PowerOn=0
Idle=1
上下出=2
檢查開始=3
上下回=4
*************************************************************************)
(*************************************************************************
異常碼
急停=1
氣缸=2
檢查NG=3
*************************************************************************)
//*************************************************************************
//本站狀態判斷
IF IndexData[2].OKFlag[2]
	OR IndexData[2].NGFlag[2] THEN
	IndexData[2].FinishFlag[2]:=TRUE;
END_IF;
//前站狀態判斷
IF  	IndexData[2].NGFlag[1] THEN
	IndexData[2].NGFlag[1]:=TRUE;
END_IF;
//本站關閉判斷
IF DisablePB[2] AND IndexData[2].FinishFlag[1] AND IndexData[2].OKFlag[1] AND NOT(IndexData[2].NGFlag[1]) THEN
	IndexData[2].OKFlag[2]:=TRUE;
END_IF;

Rtrig_test(CLK:=TestPB[2]);
//PowerOn=0
IF NOT(SystemReadyStatus AND AutoStatus AND NOT(ErrorStatus[2]) AND NOT(Error_PB_EStop)) THEN
	Autoflow:=0;
END_IF;
	//EStop異常碼
	(*IF Error_PB_Estop AND NOT(IndexData[4].FinishFlag[4]) AND IndexData[4].OkFlag[1] THEN
		IndexData[4].NGFlag[4]:=TRUE;
		IndexData[4].ErrorLog[4]:=1;
	END_IF;*)
	//Error異常碼
	(*IF ErrorStatus[4] AND NOT(IndexData[4].FinishFlag[4]) AND IndexData[4].OkFlag[1] THEN
		IndexData[4].NGFlag[4]:=TRUE;
		IndexData[4].ErrorLog[4]:=2;
	END_IF;*)
//Idle=1
IF AutoFlow=0 AND SystemReadyStatus AND AutoStatus AND NOT(ErrorStatus[2]) AND NOT(Error_PB_EStop) THEN
	AutoFlow:=1;
END_IF;

IF Autoflow=4 AND LS_S2_UpDownBack THEN
	Autoflow:=1;
END_IF;

//上下出=2
IF Autoflow=1
	AND AutoStatus
	AND NOT(DisablePB[2])
	AND LS_S2_UpDownBack
	AND (MachineRunStatus AND NOT(IndexData[2].FinishFlag[2]) AND IndexData[2].FinishFlag[1] AND IndexData[2].OKFlag[1] AND NOT(IndexData[2].NGFlag[1])
	OR Rtrig_test.Q) THEN
	Autoflow:=2;
END_IF;

//檢查開始=3
IF Autoflow=2 AND NOT(LS_S2_UpDownBack) THEN
	Autoflow:=3;
END_IF;
TON1(In:=Autoflow=3 AND LS_S2_UpDownOut, PT:=t#500ms);		//OK
TON2(In:=Autoflow=3 AND NOT(LS_S2_UpDownOut), PT:=t#2000ms);		//NG
//上下回=4
IF Autoflow=3 AND TON1.Q THEN
	IndexData[2].OKFlag[2]:=TRUE;
	IndexData[2].NGFlag[2]:=FALSE;
	Autoflow:=4;
END_IF;

IF Autoflow=3 AND TON2.Q THEN
	IndexData[2].OKFlag[2]:=FALSE;
	IndexData[2].NGFlag[2]:=TRUE;
	IndexData[2].ErrorLog[2]:=3;
	Autoflow:=4;
END_IF;

//*************************************************************************
//手動
//上下電磁閥
R_TRIG_1[0](CLK:=HMIPB_SOL_S2_UpDown AND NOT(AutoStatus));
interlockback[0]:=TRUE;
interlockout[0]:=SNR_Index AND NOT(RY_Index);
(*SET*)
IF ((R_TRIG_1[0].Q AND NOT(solstatus[0])) OR Autoflow=2) AND interlockout[0] THEN
	SOL_S2_UpDown:=TRUE;
END_IF;
(*RESET*)
IF ((R_TRIG_1[0].Q AND (solstatus[0])) OR Autoflow=4 OR Initflow=4) AND interlockback[0] THEN
	SOL_S2_UpDown:=FALSE;
END_IF;
(*STATUS*)
solstatus[0]:=SOL_S2_UpDown;
(*************************************************************************
程序名稱:第2站檢查下夾板RESET流程
作者:蔡相偉
版本,日期,版本資訊:
1.0.0		2017/11/22		初始版本

PowerOn=0
Idle=1
上下回=4
*************************************************************************)
//PowerOn=0
IF NOT(SystemReadyStatus) THEN
	Initflow:=0;
END_IF;

//Idle=1
IF Initflow=0 AND SystemReadyStatus THEN
	Initflow:=1;
END_IF;

IF Initflow=4 AND LS_S2_UpDownBack THEN
	Initflow:=1;
END_IF;

//上下回=4
F_TRIG_1(CLK:= ErrorStatus[2] OR Error_PB_Estop);
IF Initflow=1 AND (F_TRIG_1.Q OR Manual2AutoFlag) THEN
	Initflow:=4;
END_IF;
END_PROGRAM

PROGRAM prStation5
VAR
    interlockback : ARRAY[0..1] OF BOOL;
    interlockout : ARRAY[0..1] OF BOOL;
    solstatus : ARRAY[0..1] OF BOOL;
    R_TRIG_1 : ARRAY[0..1] OF R_TRIG;
    Rtrig_test : R_TRIG;
    F_TRIG_1 : F_TRIG;
    Autoflow : INT;
    Initflow : INT;
    TON1 : TON;
    TON2 : TON;
END_VAR
VAR_EXTERNAL
    IndexData : ARRAY[0..19] OF stIndexData;
    DisablePB : ARRAY[0..19] OF BOOL;
    SystemReadyStatus : BOOL;
    AutoStatus : BOOL;
    ErrorStatus : ARRAY[0..19] OF BOOL;
    Error_PB_EStop : BOOL;
    MachineRunStatus : BOOL;
    SNR_Index : BOOL;
    RY_Index : BOOL;
    Manual2AutoFlag : BOOL;
    TestPB : ARRAY[0..19] OF BOOL;
    SNR_S5_Check : BOOL;
END_VAR
(*************************************************************************
程序名稱:第5站檢查轉子組流程
作者:蔡相偉
版本,日期,版本資訊:
1.0.0		2017/11/22		初始版本

PowerOn=0
Idle=1
檢查開始=2
檢查完成=3
*************************************************************************)
(*************************************************************************
異常碼
急停=1
氣缸=2
檢查NG=3
*************************************************************************)
//*************************************************************************
//本站狀態判斷
IF IndexData[5].OKFlag[5]
	OR IndexData[5].NGFlag[5] THEN
	IndexData[5].FinishFlag[5]:=TRUE;
END_IF;
//前站狀態判斷
IF  	IndexData[5].NGFlag[4] THEN
	IndexData[5].NGFlag[5]:=TRUE;
END_IF;
//本站關閉判斷
IF DisablePB[5] AND IndexData[5].FinishFlag[4] AND IndexData[5].OKFlag[4] AND NOT(IndexData[5].NGFlag[4]) THEN
	IndexData[5].OKFlag[5]:=TRUE;
END_IF;

Rtrig_test(CLK:=TestPB[5]);
//PowerOn=0
IF NOT(SystemReadyStatus AND AutoStatus AND NOT(ErrorStatus[5]) AND NOT(Error_PB_EStop)) THEN
	Autoflow:=0;
END_IF;
	//EStop異常碼
	(*IF Error_PB_Estop AND NOT(IndexData[4].FinishFlag[4]) AND IndexData[4].OkFlag[1] THEN
		IndexData[4].NGFlag[4]:=TRUE;
		IndexData[4].ErrorLog[4]:=1;
	END_IF;*)
	//Error異常碼
	(*IF ErrorStatus[4] AND NOT(IndexData[4].FinishFlag[4]) AND IndexData[4].OkFlag[1] THEN
		IndexData[4].NGFlag[4]:=TRUE;
		IndexData[4].ErrorLog[4]:=2;
	END_IF;*)
//Idle=1
IF AutoFlow=0 AND SystemReadyStatus AND AutoStatus AND NOT(ErrorStatus[5]) AND NOT(Error_PB_EStop) THEN
	AutoFlow:=1;
END_IF;

IF Autoflow=3 AND IndexData[5].FinishFlag[5] THEN
	Autoflow:=1;
END_IF;

//檢查開始=2
IF Autoflow=1
	AND AutoStatus
	AND NOT(DisablePB[5])
	AND SNR_Index
	AND NOT(RY_Index)
	AND (MachineRunStatus AND NOT(IndexData[5].FinishFlag[5]) AND IndexData[5].FinishFlag[4] AND IndexData[5].OKFlag[4] AND NOT(IndexData[5].NGFlag[4])
	OR Rtrig_test.Q) THEN
	Autoflow:=2;
END_IF;
TON1(In:=Autoflow=2 AND SNR_S5_Check, PT:=t#500ms);		//OK
TON2(In:=Autoflow=2 AND NOT(SNR_S5_Check), PT:=t#1000ms);		//NG
//檢查完成=3
IF Autoflow=2 AND TON1.Q THEN
	IndexData[5].OKFlag[5]:=TRUE;
	IndexData[5].NGFlag[5]:=FALSE;
	Autoflow:=3;
END_IF;
IF Autoflow=2 AND TON2.Q THEN
	IndexData[5].OKFlag[5]:=FALSE;
	IndexData[5].NGFlag[5]:=TRUE;
	IndexData[5].ErrorLog[5]:=3;
	Autoflow:=3;
END_IF;
END_PROGRAM

PROGRAM prStation7
VAR
    interlockback : ARRAY[0..1] OF BOOL;
    interlockout : ARRAY[0..1] OF BOOL;
    solstatus : ARRAY[0..1] OF BOOL;
    R_TRIG_1 : ARRAY[0..1] OF R_TRIG;
    Rtrig_test : R_TRIG;
    F_TRIG_1 : F_TRIG;
    Autoflow : INT;
    Initflow : INT;
    TON1 : TON;
    TON2 : TON;
END_VAR
VAR_EXTERNAL
    IndexData : ARRAY[0..19] OF stIndexData;
    DisablePB : ARRAY[0..19] OF BOOL;
    SystemReadyStatus : BOOL;
    AutoStatus : BOOL;
    ErrorStatus : ARRAY[0..19] OF BOOL;
    Error_PB_EStop : BOOL;
    MachineRunStatus : BOOL;
    SNR_Index : BOOL;
    RY_Index : BOOL;
    Manual2AutoFlag : BOOL;
    TestPB : ARRAY[0..19] OF BOOL;
    SNR_S7_Check : BOOL;
END_VAR
(*************************************************************************
程序名稱:第7站檢查齒輪流程
作者:蔡相偉
版本,日期,版本資訊:
1.0.0		2017/11/22		初始版本

PowerOn=0
Idle=1
檢查開始=2
檢查完成=3
*************************************************************************)
(*************************************************************************
異常碼
急停=1
氣缸=2
檢查NG=3
*************************************************************************)
//*************************************************************************
//本站狀態判斷
IF IndexData[7].OKFlag[7]
	OR IndexData[7].NGFlag[7] THEN
	IndexData[7].FinishFlag[7]:=TRUE;
END_IF;
//前站狀態判斷
IF  	IndexData[7].NGFlag[6] THEN
	IndexData[7].NGFlag[7]:=TRUE;
END_IF;
//本站關閉判斷
IF DisablePB[7] AND IndexData[7].FinishFlag[6] AND IndexData[7].OKFlag[6] AND NOT(IndexData[7].NGFlag[6]) THEN
	IndexData[7].OKFlag[7]:=TRUE;
END_IF;

Rtrig_test(CLK:=TestPB[7]);
//PowerOn=0
IF NOT(SystemReadyStatus AND AutoStatus AND NOT(ErrorStatus[7]) AND NOT(Error_PB_EStop)) THEN
	Autoflow:=0;
END_IF;
	//EStop異常碼
	(*IF Error_PB_Estop AND NOT(IndexData[4].FinishFlag[4]) AND IndexData[4].OkFlag[1] THEN
		IndexData[4].NGFlag[4]:=TRUE;
		IndexData[4].ErrorLog[4]:=1;
	END_IF;*)
	//Error異常碼
	(*IF ErrorStatus[4] AND NOT(IndexData[4].FinishFlag[4]) AND IndexData[4].OkFlag[1] THEN
		IndexData[4].NGFlag[4]:=TRUE;
		IndexData[4].ErrorLog[4]:=2;
	END_IF;*)
//Idle=1
IF AutoFlow=0 AND SystemReadyStatus AND AutoStatus AND NOT(ErrorStatus[7]) AND NOT(Error_PB_EStop) THEN
	AutoFlow:=1;
END_IF;

IF Autoflow=3 AND IndexData[7].FinishFlag[7] THEN
	Autoflow:=1;
END_IF;

//檢查開始=2
IF Autoflow=1
	AND AutoStatus
	AND NOT(DisablePB[7])
	AND SNR_Index
	AND NOT(RY_Index)
	AND (MachineRunStatus AND NOT(IndexData[7].FinishFlag[7]) AND IndexData[7].FinishFlag[6] AND IndexData[7].OKFlag[6] AND NOT(IndexData[7].NGFlag[6])
	OR Rtrig_test.Q) THEN
	Autoflow:=2;
END_IF;
TON1(In:=Autoflow=2 AND SNR_S7_Check, PT:=t#500ms);		//OK
TON2(In:=Autoflow=2 AND NOT(SNR_S7_Check), PT:=t#1000ms);		//NG
//檢查完成=3
IF Autoflow=2 AND TON1.Q THEN
	IndexData[7].OKFlag[7]:=TRUE;
	IndexData[7].NGFlag[7]:=FALSE;
	Autoflow:=3;
END_IF;
IF Autoflow=2 AND TON2.Q THEN
	IndexData[7].OKFlag[7]:=FALSE;
	IndexData[7].NGFlag[7]:=TRUE;
	IndexData[7].ErrorLog[7]:=3;
	Autoflow:=3;
END_IF;
END_PROGRAM

PROGRAM prStation9
VAR
    interlockback : ARRAY[0..1] OF BOOL;
    interlockout : ARRAY[0..1] OF BOOL;
    solstatus : ARRAY[0..1] OF BOOL;
    R_TRIG_1 : ARRAY[0..1] OF R_TRIG;
    Rtrig_test : R_TRIG;
    F_TRIG_1 : F_TRIG;
    Autoflow : INT;
    Initflow : INT;
    TON1 : TON;
    TON2 : TON;
END_VAR
VAR_EXTERNAL
    IndexData : ARRAY[0..19] OF stIndexData;
    DisablePB : ARRAY[0..19] OF BOOL;
    SystemReadyStatus : BOOL;
    AutoStatus : BOOL;
    ErrorStatus : ARRAY[0..19] OF BOOL;
    Error_PB_EStop : BOOL;
    MachineRunStatus : BOOL;
    SNR_Index : BOOL;
    RY_Index : BOOL;
    Manual2AutoFlag : BOOL;
    TestPB : ARRAY[0..19] OF BOOL;
    SNR_S9_Check : BOOL;
END_VAR
(*************************************************************************
程序名稱:第9站檢查卡子流程
作者:蔡相偉
版本,日期,版本資訊:
1.0.0		2017/11/22		初始版本

PowerOn=0
Idle=1
檢查開始=2
檢查完成=3
*************************************************************************)
(*************************************************************************
異常碼
急停=1
氣缸=2
檢查NG=3
*************************************************************************)
//*************************************************************************
//本站狀態判斷
IF IndexData[9].OKFlag[9]
	OR IndexData[9].NGFlag[9] THEN
	IndexData[9].FinishFlag[9]:=TRUE;
END_IF;
//前站狀態判斷
IF  	IndexData[9].NGFlag[8] THEN
	IndexData[9].NGFlag[9]:=TRUE;
END_IF;
//本站關閉判斷
IF DisablePB[9] AND IndexData[9].FinishFlag[8] AND IndexData[9].OKFlag[8] AND NOT(IndexData[9].NGFlag[8]) THEN
	IndexData[9].OKFlag[9]:=TRUE;
END_IF;

Rtrig_test(CLK:=TestPB[9]);
//PowerOn=0
IF NOT(SystemReadyStatus AND AutoStatus AND NOT(ErrorStatus[9]) AND NOT(Error_PB_EStop)) THEN
	Autoflow:=0;
END_IF;
	//EStop異常碼
	(*IF Error_PB_Estop AND NOT(IndexData[4].FinishFlag[4]) AND IndexData[4].OkFlag[1] THEN
		IndexData[4].NGFlag[4]:=TRUE;
		IndexData[4].ErrorLog[4]:=1;
	END_IF;*)
	//Error異常碼
	(*IF ErrorStatus[4] AND NOT(IndexData[4].FinishFlag[4]) AND IndexData[4].OkFlag[1] THEN
		IndexData[4].NGFlag[4]:=TRUE;
		IndexData[4].ErrorLog[4]:=2;
	END_IF;*)
//Idle=1
IF AutoFlow=0 AND SystemReadyStatus AND AutoStatus AND NOT(ErrorStatus[9]) AND NOT(Error_PB_EStop) THEN
	AutoFlow:=1;
END_IF;

IF Autoflow=3 AND IndexData[9].FinishFlag[9] THEN
	Autoflow:=1;
END_IF;

//檢查開始=2
IF Autoflow=1
	AND AutoStatus
	AND NOT(DisablePB[9])
	AND SNR_Index
	AND NOT(RY_Index)
	AND (MachineRunStatus AND NOT(IndexData[9].FinishFlag[9]) AND IndexData[9].FinishFlag[8] AND IndexData[9].OKFlag[8] AND NOT(IndexData[9].NGFlag[8])
	OR Rtrig_test.Q) THEN
	Autoflow:=2;
END_IF;
TON1(In:=Autoflow=2 AND SNR_S9_Check, PT:=t#500ms);		//OK
TON2(In:=Autoflow=2 AND NOT(SNR_S9_Check), PT:=t#1000ms);		//NG
//檢查完成=3
IF Autoflow=2 AND TON1.Q THEN
	IndexData[9].OKFlag[9]:=TRUE;
	IndexData[9].NGFlag[9]:=FALSE;
	Autoflow:=3;
END_IF;
IF Autoflow=2 AND TON2.Q THEN
	IndexData[9].OKFlag[9]:=FALSE;
	IndexData[9].NGFlag[9]:=TRUE;
	IndexData[9].ErrorLog[9]:=3;
	Autoflow:=3;
END_IF;
END_PROGRAM

FUNCTION_BLOCK fbErrorDouble
VAR
    TON_1 : TON;
    TON_2 : TON;
END_VAR
VAR_INPUT
    bAutoStatus : BOOL;
    bResetPB : BOOL;
    bBackLS : BOOL;
    bOutLS : BOOL;
    bBackSOL : BOOL;
    bOutSOL : BOOL;
END_VAR
VAR_OUTPUT
    bErrorStatus_Back : BOOL;
    bErrorStatus_Out : BOOL;
END_VAR
IF bAutoStatus AND NOT(bResetPB) THEN
	(*歸磁簧開關*)
	TON_1(IN:=bBackSOL AND NOT(bBackLS), PT:=t#5s);
	IF TON_1.Q THEN
		bErrorStatus_Back:=TRUE;
	END_IF;
	(*出磁簧開關*)
	TON_2(IN:=bOutSOL AND NOT(bOutLS), PT:=t#5s);
	IF TON_2.Q THEN
		bErrorStatus_Out:=TRUE;
	END_IF;
END_IF;
IF bResetPB THEN
	bErrorStatus_Back:=FALSE;
	bErrorStatus_Out:=FALSE;
END_IF;
END_FUNCTION_BLOCK

FUNCTION_BLOCK fbErrorSingle
VAR
    TON_1 : TON;
    TON_2 : TON;
END_VAR
VAR_INPUT
    bAutoStatus : BOOL;
    bResetPB : BOOL;
    bSOL : BOOL;
    bBackLS : BOOL;
    bOutLS : BOOL;
END_VAR
VAR_OUTPUT
    bErrorStatus_Back : BOOL;
    bErrorStatus_Out : BOOL;
END_VAR
IF bAutoStatus AND NOT(bResetPB) THEN
	(*歸磁簧開關*)
	TON_1(IN:=(NOT(bSOL) AND NOT(bBackLS)) OR ((bSOL) AND bBackLS), PT:=t#5s);
	IF TON_1.Q THEN
		bErrorStatus_Back:=TRUE;
	END_IF;
	(*出磁簧開關*)
	TON_2(IN:=(NOT(bSOL) AND (bOutLS)) OR ((bSOL) AND NOT(bOutLS)), PT:=t#5s);
	IF TON_2.Q THEN
		bErrorStatus_Out:=TRUE;
	END_IF;
END_IF;
IF bResetPB THEN
	bErrorStatus_Back:=FALSE;
	bErrorStatus_Out:=FALSE;
END_IF;
END_FUNCTION_BLOCK